TYPE ST_MC_Status :
STRUCT
	Status	: BOOL;
	Done	: BOOL;
	Busy	: BOOL;
	Error	: BOOL;
	Active	: BOOL;
	CmdAborted	: BOOL;
	InVelocity	: BOOL;
	ErrorID	: UDINT;
	
END_STRUCT
END_TYPE

(* stored: Version 1.1.0.1, ProductVersion 3.1.4024.12
   DUT ST_MC_Status: Id {0905a629-31d8-4bf3-8dd0-cfdd05ffed33} *)
